// SIMATIC S7-200 project (STEP 7-Micro/WIN), CPU 224XP REL 02.01

SYMBOL_TABLE USUARIO1
P_I_SEGURIDAD    I0.0
P_D_SEGURIDAD    I0.1
C_F_C            Q0.0
F_C_1            Q0.1
F_C_2            Q0.2
F_C_3            Q0.3
F_C_4            Q0.4
C_G              Q0.5
GUILLOTINA       Q0.6
END_SYMBOL_TABLE

SYMBOL_TABLE Símbolos S7-200
Primer_ciclo_ON  SM0.1    // ON sólo en el primer ciclo
END_SYMBOL_TABLE

ORGANIZATION_BLOCK PRINCIPAL:OB1
TITLE=COMENTARIOS DEL PROGRAMA
BEGIN
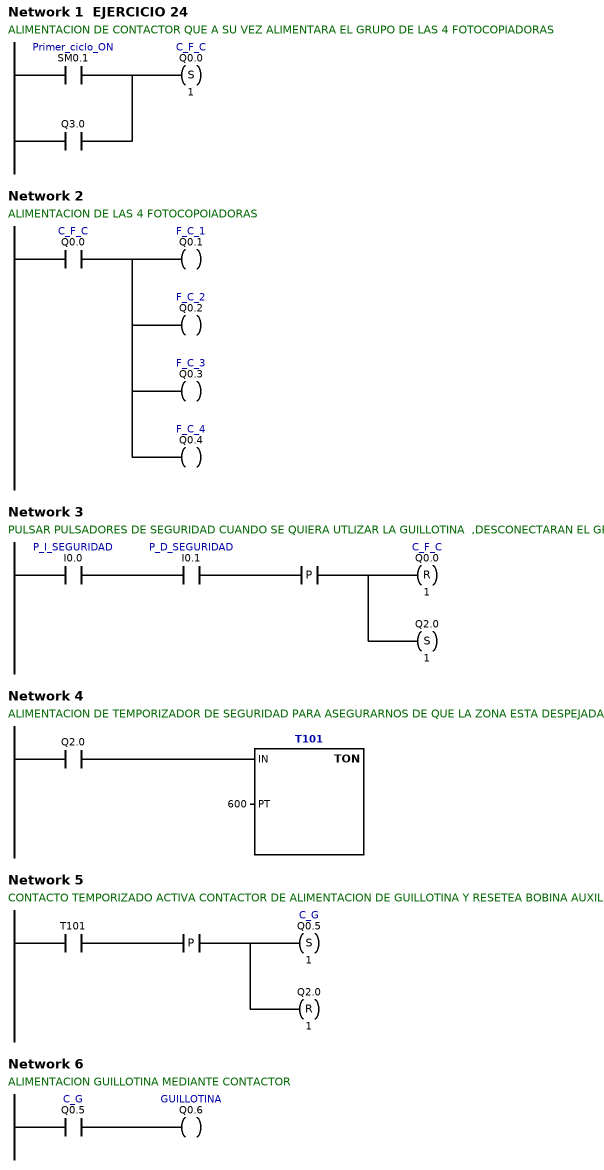
Network 1 // EJERCICIO 24
// ALIMENTACION DE CONTACTOR QUE A SU VEZ ALIMENTARA EL GRUPO DE LAS 4 FOTOCOPIADORAS
LD     Primer_ciclo_ON:SM0.1
O      Q3.0
S      C_F_C:Q0.0, 1
Network 2
// ALIMENTACION DE LAS 4 FOTOCOPOIADORAS 
LD     C_F_C:Q0.0
=      F_C_1:Q0.1
=      F_C_2:Q0.2
=      F_C_3:Q0.3
=      F_C_4:Q0.4
Network 3
// PULSAR PULSADORES DE SEGURIDAD CUANDO SE QUIERA UTLIZAR LA GUILLOTINA  ,DESCONECTARAN EL GRUPO DE FOTOCOPIADORAS 
LD     P_I_SEGURIDAD:I0.0
A      P_D_SEGURIDAD:I0.1
EU
R      C_F_C:Q0.0, 1
S      Q2.0, 1
Network 4
// ALIMENTACION DE TEMPORIZADOR DE SEGURIDAD PARA ASEGURARNOS DE QUE LA ZONA ESTA DESPEJADA
LD     Q2.0
TON    T101, 600
Network 5
// CONTACTO TEMPORIZADO ACTIVA CONTACTOR DE ALIMENTACION DE GUILLOTINA Y RESETEA BOBINA AUXILIAR
LD     T101
EU
S      C_G:Q0.5, 1
R      Q2.0, 1
Network 6
// ALIMENTACION GUILLOTINA MEDIANTE CONTACTOR 
LD     C_G:Q0.5
=      GUILLOTINA:Q0.6
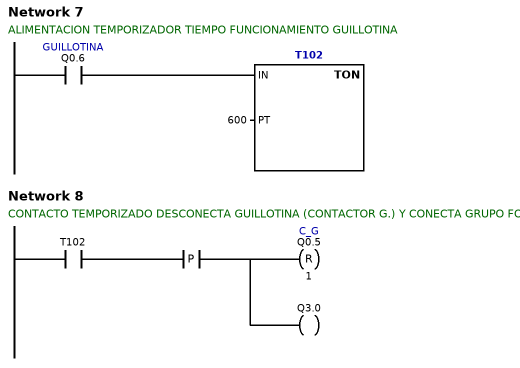
Network 7
// ALIMENTACION TEMPORIZADOR TIEMPO FUNCIONAMIENTO GUILLOTINA
LD     GUILLOTINA:Q0.6
TON    T102, 600
Network 8
// CONTACTO TEMPORIZADO DESCONECTA GUILLOTINA (CONTACTOR G.) Y CONECTA GRUPO FOTOCOPIADORAS  (CN¡ONTACTOR F.C)
LD     T102
EU
R      C_G:Q0.5, 1
=      Q3.0
END_ORGANIZATION_BLOCK
